FUNCTION TryConvert_LREAL_TO_BOOL : BOOL
VAR_INPUT
	in : LREAL;
	out : REFERENCE TO BOOL;
END_VAR

out := LREAL_TO_BOOL(in);
TryConvert_LREAL_TO_BOOL := TRUE;

END_FUNCTION

(* stored: Version 1.1.0.1, ProductVersion 3.1.4024.12
   POU TryConvert_LREAL_TO_BOOL: Id {8f0a0880-9858-4f5a-a389-a8e531756790}, SpecialFunc None *)
